Staubli VAL3: DeplacementInit.pgx

program DeplacementInit()
begin
  movej(jInitial, tTool, mDeplacement)
end
